{attribute 'linkalways'} 
{attribute 'no_explicit_call' := 'This FB is a CLASS and must be accessed using methods or properties'}
{attribute 'enable_dynamic_creation'}
FUNCTION_BLOCK _ETcVn2dCodeSearchStrategy EXTENDS EnumDatatypeBase
VAR
	localData : ETcVn2dCodeSearchStrategy;
	activeData : REFERENCE TO ETcVn2dCodeSearchStrategy;
	enumBaseDatatype : _UDINT(localData);
END_VAR

METHOD PRIVATE AddLocalEnumeration
VAR_INPUT
	Enumeration : T_MAXSTRING;
	Value : ETcVn2dCodeSearchStrategy;
END_VAR
AddEnumeration(Enumeration, Value);
END_METHOD

PROPERTY PUBLIC Address : PVOID
GET
Address := ADR(activeData);
END_GET
END_PROPERTY

METHOD PUBLIC ClearReference
VAR_INPUT
END_VAR
activeData REF= localData;
SetBaseDatatypeReference();
END_METHOD

METHOD PUBLIC Clone : I_Datatype
VAR
    pClone : POINTER TO _ETcVn2dCodeSearchStrategy;
END_VAR
pClone := __NEW(_ETcVn2dCodeSearchStrategy(InitialValue := Value));
Clone := pClone^;
END_METHOD

METHOD FB_init : BOOL
VAR_INPUT
	bInitRetains : BOOL; // if TRUE, the retain variables are initialized (warm start / cold start)
	bInCopyCode : BOOL;  // if TRUE, the instance afterwards gets moved into the copy code (online change)
	InitialValue : ETcVn2dCodeSearchStrategy;
END_VAR
localData := InitialValue;
AddBaseDatatype(enumBaseDatatype);
ClearReference();

AddLocalEnumeration('TCVN_CSS_DEFAULT', ETcVn2dCodeSearchStrategy.TCVN_CSS_DEFAULT);
AddLocalEnumeration('TCVN_CSS_FIRST_FLIPPED', ETcVn2dCodeSearchStrategy.TCVN_CSS_FIRST_FLIPPED);
AddLocalEnumeration('TCVN_CSS_FIRST_INVERTED', ETcVn2dCodeSearchStrategy.TCVN_CSS_FIRST_INVERTED);
AddLocalEnumeration('TCVN_CSS_FIRST_NOT_FLIPPED', ETcVn2dCodeSearchStrategy.TCVN_CSS_FIRST_NOT_FLIPPED);
AddLocalEnumeration('TCVN_CSS_FIRST_NOT_INVERTED', ETcVn2dCodeSearchStrategy.TCVN_CSS_FIRST_NOT_INVERTED);
AddLocalEnumeration('TCVN_CSS_ONLY_FLIPPED', ETcVn2dCodeSearchStrategy.TCVN_CSS_ONLY_FLIPPED);
AddLocalEnumeration('TCVN_CSS_ONLY_INVERTED', ETcVn2dCodeSearchStrategy.TCVN_CSS_ONLY_INVERTED);
AddLocalEnumeration('TCVN_CSS_ONLY_NOT_FLIPPED', ETcVn2dCodeSearchStrategy.TCVN_CSS_ONLY_NOT_FLIPPED);
AddLocalEnumeration('TCVN_CSS_ONLY_NOT_INVERTED', ETcVn2dCodeSearchStrategy.TCVN_CSS_ONLY_NOT_INVERTED);
END_METHOD

PROPERTY PUBLIC Identifier : T_MAXSTRING
GET
Identifier := 'ETcVn2dCodeSearchStrategy';
END_GET
END_PROPERTY

METHOD IsEnumeratorValueEqual : BOOL
VAR_INPUT
	Enumerator : I_KeyValueForwardEnumerator;
END_VAR
VAR
	storedValue : ETcVn2dCodeSearchStrategy;
END_VAR
IF NOT Enumerator.TryGet(storedValue) THEN
	RETURN;
END_IF

IsEnumeratorValueEqual := storedValue = activeData;
END_METHOD

METHOD PUBLIC MakeReferenceTo
VAR_INPUT
	ReferenceTarget : REFERENCE TO ETcVn2dCodeSearchStrategy;
END_VAR
activeData REF= ReferenceTarget;
SetBaseDatatypeReference();
END_METHOD

METHOD PROTECTED SetBaseDatatypeReference
VAR_INPUT
END_VAR
enumBaseDatatype.MakeReferenceTo(activeData);
END_METHOD

PROPERTY PUBLIC Size : UDINT
GET
Size := SIZEOF(activeData);
END_GET
END_PROPERTY

METHOD TryMakeReferenceTo : BOOL
VAR_INPUT
	Target : I_Datatype;
END_VAR
VAR
	targetAsEnum : I_EnumDatatype;
	pTargetData : POINTER TO ETcVn2dCodeSearchStrategy;
END_VAR
IF NOT Target.TryResolveAsEnumDatatype(targetAsEnum) THEN
	RETURN;
END_IF

IF targetAsEnum.Identifier <> Identifier THEN
	RETURN;
END_IF

pTargetData := Target.Address;
activeData REF= pTargetData^;
SetBaseDatatypeReference();
TryMakeReferenceTo := TRUE;
END_METHOD

PROPERTY PUBLIC Value : ETcVn2dCodeSearchStrategy
GET
Value := activeData;
END_GET
SET
activeData := Value;
END_SET
END_PROPERTY

END_FUNCTION_BLOCK

(* stored: Version 1.1.0.1, ProductVersion 3.1.4024.12
   POU _ETcVn2dCodeSearchStrategy: Id {c1ea101a-c1de-0219-3556-045633e43bb3}, SpecialFunc None
   Folder Constructor: Id {e8cc02fa-501d-0e1f-131c-4ee069a2762f}
   Folder Private: Id {6c4d79f9-c5a2-0c20-1f88-4642fbdbda3d}
   Folder Protected: Id {8af1eaa5-6ab0-0b60-0ee1-5529ca2e2225}
   Method AddLocalEnumeration: Id {c8e4c393-36f5-0e56-0d70-8f44f1723af9}
   Property Address: Id {462e3f31-b3af-0f4a-2f1a-bee76a8337e7}
   Get Get: Id {fc6961e5-a1f2-08ef-2953-d6d226d6bbfb}
   Method ClearReference: Id {e11f4e1b-094c-0e00-03d1-38a196054a3d}
   Method Clone: Id {eddfdfc1-07b9-0ef0-2646-ea7a753545bc}
   Method FB_init: Id {14f23aaa-7e1d-0aed-2320-3c82011d0332}
   Property Identifier: Id {c949c30e-73d3-0f27-15c6-52067e56d6c7}
   Get Get: Id {ccf77c72-b6c1-0504-0103-ad5c53df9cf6}
   Method IsEnumeratorValueEqual: Id {f06ad732-9339-0d9b-3687-86118de551cf}
   Method MakeReferenceTo: Id {fe6456c4-4cfe-0019-0828-1dc718ad9de8}
   Method SetBaseDatatypeReference: Id {8901f5e2-f941-018b-3cf7-92107684f571}
   Property Size: Id {cdf96285-acc8-0fcc-38d8-68ce4e29c4c9}
   Get Get: Id {0897d154-4342-065c-37f5-f95683d04173}
   Method TryMakeReferenceTo: Id {5454661e-b96e-0b83-3e8a-4d17dddb8cf5}
   Property Value: Id {24ef3cd8-2bc5-0b8b-11c2-567a37edde5a}
   Get Get: Id {cce7ea5e-c79e-08a7-0b26-046d8b7f7626}
   Set Set: Id {2609190e-65bb-0de2-3f58-4e8a06fae32f} *)
